// LS Electric XG5000 project: 7_모타증감회로
// PLC NewPLC
// module base 0 slot 0: 입출력 모듈:XBC-DN/DP14E (DC 24V 입력 8점, 트랜지스터 출력 6점)

PROGRAM NewProgram (task: 스캔 프로그램)

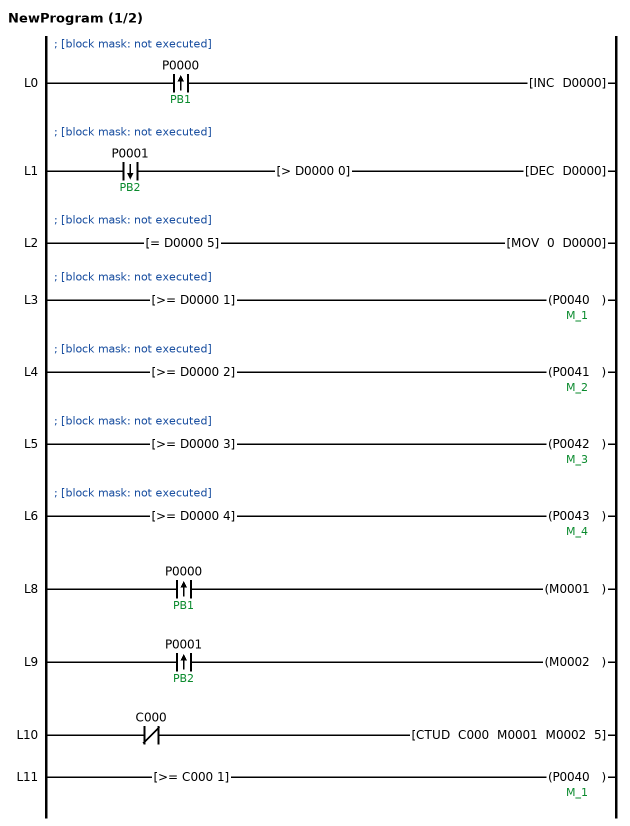
; L0 (block mask: not executed)
LOADP     P0000	// PB1
INC       D0000
; L1 (block mask: not executed)
LOADN     P0001	// PB2
AND>      D0000 0
DEC       D0000
; L2 (block mask: not executed)
LOAD=     D0000 5
MOV       0 D0000
; L3 (block mask: not executed)
LOAD>=    D0000 1
OUT       P0040	// M_1
; L4 (block mask: not executed)
LOAD>=    D0000 2
OUT       P0041	// M_2
; L5 (block mask: not executed)
LOAD>=    D0000 3
OUT       P0042	// M_3
; L6 (block mask: not executed)
LOAD>=    D0000 4
OUT       P0043	// M_4
; L8
LOADP     P0000	// PB1
OUT       M0001
; L9
LOADP     P0001	// PB2
OUT       M0002
; L10
LOAD NOT  C000
CTUD      C000 M0001 M0002 5
; L11
LOAD>=    C000 1
OUT       P0040	// M_1

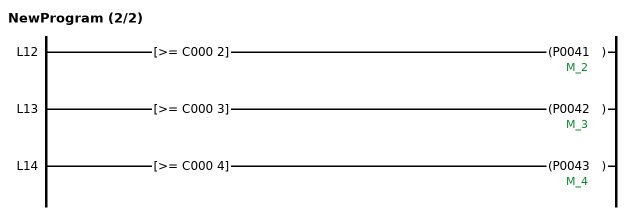
; L12
LOAD>=    C000 2
OUT       P0041	// M_2
; L13
LOAD>=    C000 3
OUT       P0042	// M_3
; L14
LOAD>=    C000 4
OUT       P0043	// M_4